(*
typedef struct _PTPTime
{
	ULONGLONG internal;
	ULONGLONG external;
	bool not_connected;
	bool update_toggle;
	LONGLONG dcTcOffset;
} PTPTime, *PPTPTime;
*)
TYPE T_PTP_TIME :
STRUCT
END_STRUCT
END_TYPE

(* stored: Version 1.1.0.1, ProductVersion 3.1.4022.9
   DUT T_PTP_TIME: Id {18e20439-7c75-402f-a355-d930409c54dd} *)
